// TIA Portal V19 export
VAR_GLOBAL   // PLC tag table "U2Em0_input"
END_VAR
VAR_GLOBAL CONSTANT   // user constants
   U2EM0_NO_OF_AXES : USInt := 1;   // Starts with 1. E.g., the value 4 means that 4 axes exist.
   U2EM0_JOB1 : DInt := 1;   // ID for Job
END_VAR
